// TIA Portal V20 export
DATA_BLOCK "DB_AnalogInputs"   // DB2200
// stored: AutoNumber false, InstanceOfName FB_AnalogInputs, InstanceOfType FB
"FB_AnalogInputs"
   // VAR
   //    sLaserPowerMeter : "FB_AnalogInput";
   //    sAxisB_ClampingPart : "FB_AnalogInput";
   //    sLaserAirPressureProcess : "FB_AnalogInput";
   //    sInletAirPressure : "FB_AnalogInput";
   //    sAmbiantTemperature : "FB_AnalogInput";
   //    sMachineTemperature : "FB_AnalogInput";
   //    sCold_WaterTemperatureInput : "FB_AnalogInput";
   //    sCold_WaterTemperatureOutput : "FB_AnalogInput";
   //    sX_AxisTemperaturePT1000 : "FB_AnalogInput";
   //    sY_AxisTemperaturePT1000 : "FB_AnalogInput";
   //    sX_AxisTemperaturePTC : "FB_AnalogInput";
   //    sY_AxisTemperaturePTC : "FB_AnalogInput";
   //    sNozzleOverpressure : "FB_AnalogInput";
   //    sOpticalPathOverpressure : "FB_AnalogInput";
   //    sLaserHeadOverpressure : "FB_AnalogInput";
   //    sZLAxisOverpressure : "FB_AnalogInput";
   //    sXYAxisOverpressure : "FB_AnalogInput";
   //    sLeftAspiration : "FB_AnalogInput";
   //    sRightAspiration : "FB_AnalogInput";
   //    sFreeIW458 : "FB_AnalogInput";
   //    sClimTemperature : "FB_AnalogInput";
   //    sFreeIW482 : "FB_AnalogInput";
   //    sFreeIW484 : "FB_AnalogInput";
   //    sFreeIW486 : "FB_AnalogInput";
   //    sSensorControllerStation1 : "FB_AnalogInput";
   //    sCabinetTemperature : "FB_AnalogInput";
   //    sFreeIW464 : "FB_AnalogInput";
   //    sFreeIW466 : "FB_AnalogInput";
   // END_VAR
BEGIN
END_DATA_BLOCK
